// TIA Portal V17 export
// export: Created 2022-07-20T06:59:37.1006069Z, ExportSetting WithDefaults, DisplayName Totally Integrated Automation Portal, DisplayVersion V17, DisplayName TIA Portal Openness, DisplayVersion V17, DisplayName TIA Portal Version Control Interface, DisplayVersion V17, DisplayName SINAMICS Startdrive Advanced, DisplayVersion V17, DisplayName SINAMICS Startdrive G130, G150, S120, S150, SINAMICS MV, S210, DisplayVersion V17, DisplayName SINAMICS Startdrive G110M, G120, G120C, G120D, G120P, G115D, DisplayVersion V17, DisplayName STEP 7 Professional, DisplayVersion V17, DisplayName STEP 7 Safety, DisplayVersion V17, DisplayName WinCC Advanced, DisplayVersion V17
FUNCTION_BLOCK "FB10003_Pulse"   // FB10003, LAD
TITLE = FB10003_OnePulse
{ S7_Optimized_Access := 'TRUE' }
AUTHOR : Anirouddh
FAMILY : 1000x_SYSTEM
VERSION : 1.0
// Release note : 
// 1.0 - Feature developped
// stored: AutoNumber false, IsIECCheckEnabled false, IsRetainMemResEnabled false, MemoryReserve 100, SetENOAutomatically false, UDAEnableTagReadback false
   VAR_INPUT
      CLK : Bool;
      PT : Time;
   END_VAR
   VAR_OUTPUT
      ET : Time;
   END_VAR
   VAR_IN_OUT
      Q : Bool;
   END_VAR
   VAR
      R_TRIG_Signal : R_TRIG;
      TON_Pulse : TON_TIME;
   END_VAR
BEGIN

REGION Network 1 (SCL): Edge Signals & Timers
   REGION EDGE SIGNALS
       //Signal To Start The Pulse
       #R_TRIG_Signal(CLK := #CLK);
   END_REGION

   REGION TIMERS
       //Duration Of The Pulse
       #TON_Pulse(IN := #Q,
                  PT := #PT,
                  ET => #ET);
   END_REGION
END_REGION

REGION Network 2 (SCL): Pulse Generation
   IF #R_TRIG_Signal.Q THEN
       #Q := TRUE;
   ELSIF #TON_Pulse.Q THEN
       #Q := FALSE;
   END_IF;
END_REGION
END_FUNCTION_BLOCK
